FUNCTION_BLOCK MotorS_HMI (* Service Interface Function Block Type *)
  (* Standard: 61499-2 *)
  (* Version 0.0, 6/2/2026, Schneider Electric, template *)
  PACKAGE SE.Nereda;
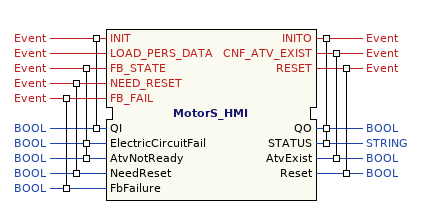
  EVENT_INPUT
    INIT WITH QI;
    LOAD_PERS_DATA;
    FB_STATE WITH ElectricCircuitFail, AtvNotReady;
    NEED_RESET WITH NeedReset;
    FB_FAIL WITH FbFailure;
  END_EVENT
  EVENT_OUTPUT
    INITO WITH QO, STATUS;
    CNF_ATV_EXIST WITH AtvExist;
    RESET WITH Reset;
  END_EVENT
  VAR_INPUT
    QI : BOOL;
    ElectricCircuitFail : BOOL;
    AtvNotReady : BOOL;
    NeedReset : BOOL;
    FbFailure : BOOL;
  END_VAR
  VAR_OUTPUT
    QO : BOOL; (* Event Output Qualifier *)
    STATUS : STRING; (* Service Status *)
    AtvExist : BOOL;
    Reset : BOOL;
  END_VAR
  SERVICE /
    SEQUENCE 
    END_SEQUENCE
  END_SERVICE
END_FUNCTION_BLOCK
